NETWORK
TITLE = CALL SFC PH_EMC2_CHARGE if CHARGE running
//------------------------------------------------------------------------//
// SFC CALL   SFC CALL   SFC CALL   SFC CALL   SFC CALL   SFC CALL   SFC  //
//                                                                        //
// Call the SFC function if this is the running substate. This has to be  //
// called even if the block is not running so the SFC can process all     //
// commmands:                                                             //
//------------------------------------------------------------------------//
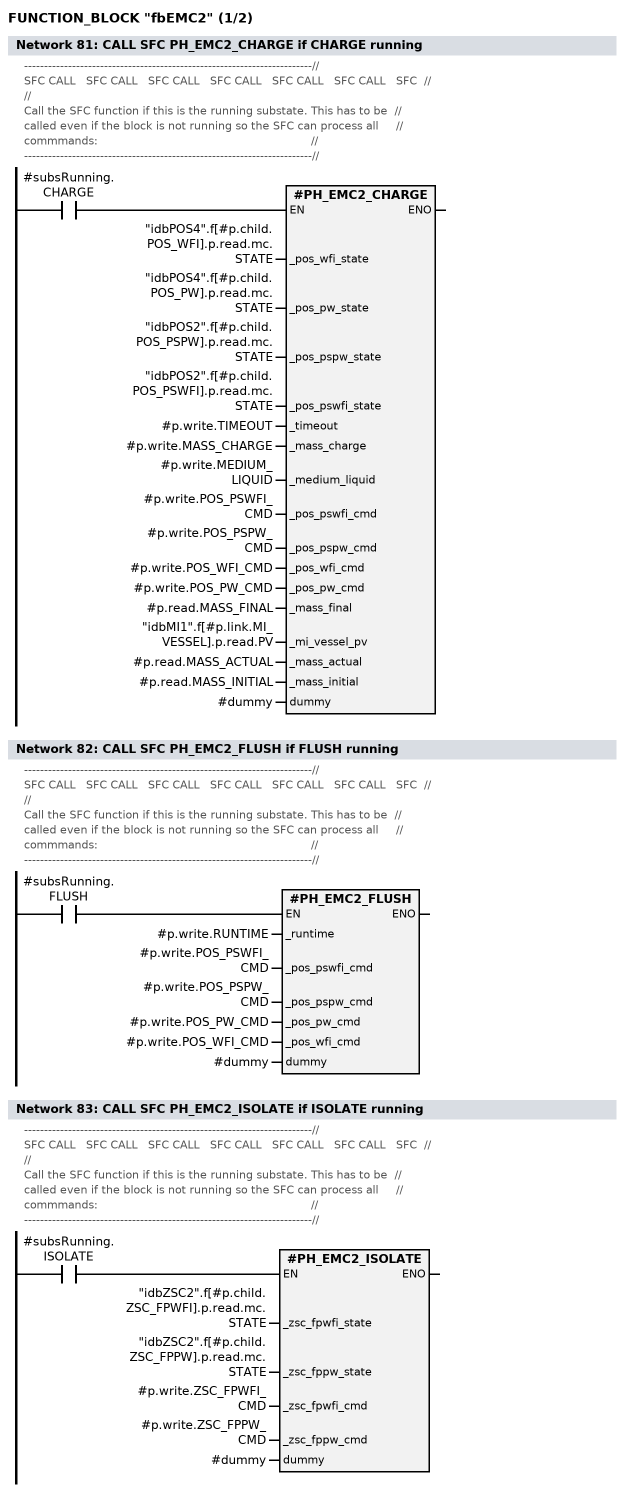
      A #subsRunning.CHARGE;
      JCN _notSFC_1_CHARGE;
      CALL #PH_EMC2_CHARGE
      (  _pos_wfi_state              := "idbPOS4".f[#p.child.POS_WFI].p.read.mc.STATE ,
         _pos_pw_state               := "idbPOS4".f[#p.child.POS_PW].p.read.mc.STATE ,
         _pos_pspw_state             := "idbPOS2".f[#p.child.POS_PSPW].p.read.mc.STATE ,
         _pos_pswfi_state            := "idbPOS2".f[#p.child.POS_PSWFI].p.read.mc.STATE ,
         _timeout                    := #p.write.TIMEOUT ,
         _mass_charge                := #p.write.MASS_CHARGE ,
         _medium_liquid              := #p.write.MEDIUM_LIQUID ,
         _pos_pswfi_cmd              := #p.write.POS_PSWFI_CMD ,
         _pos_pspw_cmd               := #p.write.POS_PSPW_CMD ,
         _pos_wfi_cmd                := #p.write.POS_WFI_CMD ,
         _pos_pw_cmd                 := #p.write.POS_PW_CMD ,
         _mass_final                 := #p.read.MASS_FINAL ,
         _mi_vessel_pv               := "idbMI1".f[#p.link.MI_VESSEL].p.read.PV ,
         _mass_actual                := #p.read.MASS_ACTUAL ,
         _mass_initial               := #p.read.MASS_INITIAL ,
         dummy                       := #dummy
      );
_notSFC_1_CHARGE:      NOP 0;
NETWORK
TITLE = CALL SFC PH_EMC2_FLUSH if FLUSH running
//------------------------------------------------------------------------//
// SFC CALL   SFC CALL   SFC CALL   SFC CALL   SFC CALL   SFC CALL   SFC  //
//                                                                        //
// Call the SFC function if this is the running substate. This has to be  //
// called even if the block is not running so the SFC can process all     //
// commmands:                                                             //
//------------------------------------------------------------------------//
      A #subsRunning.FLUSH;
      JCN _notSFC_1_FLUSH;
      CALL #PH_EMC2_FLUSH
      (  _runtime                    := #p.write.RUNTIME ,
         _pos_pswfi_cmd              := #p.write.POS_PSWFI_CMD ,
         _pos_pspw_cmd               := #p.write.POS_PSPW_CMD ,
         _pos_pw_cmd                 := #p.write.POS_PW_CMD ,
         _pos_wfi_cmd                := #p.write.POS_WFI_CMD ,
         dummy                       := #dummy
      );
_notSFC_1_FLUSH:      NOP 0;
NETWORK
TITLE = CALL SFC PH_EMC2_ISOLATE if ISOLATE running
//------------------------------------------------------------------------//
// SFC CALL   SFC CALL   SFC CALL   SFC CALL   SFC CALL   SFC CALL   SFC  //
//                                                                        //
// Call the SFC function if this is the running substate. This has to be  //
// called even if the block is not running so the SFC can process all     //
// commmands:                                                             //
//------------------------------------------------------------------------//
      A #subsRunning.ISOLATE;
      JCN _notSFC_1_ISOLATE;
      CALL #PH_EMC2_ISOLATE
      (  _zsc_fpwfi_state            := "idbZSC2".f[#p.child.ZSC_FPWFI].p.read.mc.STATE ,
         _zsc_fppw_state             := "idbZSC2".f[#p.child.ZSC_FPPW].p.read.mc.STATE ,
         _zsc_fpwfi_cmd              := #p.write.ZSC_FPWFI_CMD ,
         _zsc_fppw_cmd               := #p.write.ZSC_FPPW_CMD ,
         dummy                       := #dummy
      );
_notSFC_1_ISOLATE:      NOP 0;
NETWORK
TITLE = CALL SFC PH_EMC2_SETUP if SETUP running
//------------------------------------------------------------------------//
// SFC CALL   SFC CALL   SFC CALL   SFC CALL   SFC CALL   SFC CALL   SFC  //
//                                                                        //
// Call the SFC function if this is the running substate. This has to be  //
// called even if the block is not running so the SFC can process all     //
// commmands:                                                             //
//------------------------------------------------------------------------//
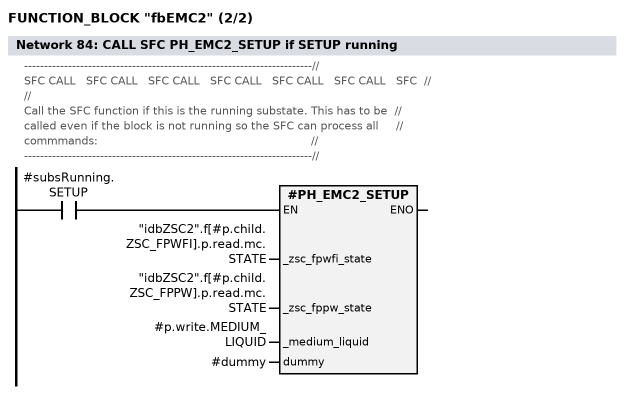
      A #subsRunning.SETUP;
      JCN _notSFC_1_SETUP;
      CALL #PH_EMC2_SETUP
      (  _zsc_fpwfi_state            := "idbZSC2".f[#p.child.ZSC_FPWFI].p.read.mc.STATE ,
         _zsc_fppw_state             := "idbZSC2".f[#p.child.ZSC_FPPW].p.read.mc.STATE ,
         _medium_liquid              := #p.write.MEDIUM_LIQUID ,
         dummy                       := #dummy
      );
_notSFC_1_SETUP:      NOP 0;

NETWORK
TITLE = Check if any Child state does not match the command
//------------------------------------------------------------------------//
// CHILD FLOWPATH STATE MISMATCH   CHILD FLOWPATH STATE MISMATCH   CHILD  //
//                                                                        //
// Check if any child flowpath device state does not match the command    //
// from this parent block if the child state grace period timer has       //
// expired. Stop checking if the first child state mismatch found:        //
//------------------------------------------------------------------------//
      A(;
      O(;
      A "alwaysHigh";
      A "idbPOS2".f[#p.child.POS_PSPW].p.write.mc.ARMED;
      A "idbPOS2".f[#p.child.POS_PSPW].p.read.mc.FLOWPATH;
      A(;
      L "idbPOS2".f[#p.child.POS_PSPW].p.read.mc.STATE;
      L #childReqCMD.POS_PSPW;
      <>I;
      );
      );
      O(;
      A "alwaysHigh";
      A "idbPOS2".f[#p.child.POS_PSWFI].p.write.mc.ARMED;
      A "idbPOS2".f[#p.child.POS_PSWFI].p.read.mc.FLOWPATH;
      A(;
      L "idbPOS2".f[#p.child.POS_PSWFI].p.read.mc.STATE;
      L #childReqCMD.POS_PSWFI;
      <>I;
      );
      );
      O(;
      A "alwaysHigh";
      A "idbPOS4".f[#p.child.POS_PW].p.write.mc.ARMED;
      A "idbPOS4".f[#p.child.POS_PW].p.read.mc.FLOWPATH;
      A(;
      L "idbPOS4".f[#p.child.POS_PW].p.read.mc.STATE;
      L #childReqCMD.POS_PW;
      <>I;
      );
      );
      O(;
      A "alwaysHigh";
      A "idbPOS4".f[#p.child.POS_WFI].p.write.mc.ARMED;
      A "idbPOS4".f[#p.child.POS_WFI].p.read.mc.FLOWPATH;
      A(;
      L "idbPOS4".f[#p.child.POS_WFI].p.read.mc.STATE;
      L #childReqCMD.POS_WFI;
      <>I;
      );
      );
      O(;
      A "alwaysHigh";
      A "idbZSC2".f[#p.child.ZSC_FPINLET].p.write.mc.ARMED;
      A "idbZSC2".f[#p.child.ZSC_FPINLET].p.read.mc.FLOWPATH;
      A(;
      L "idbZSC2".f[#p.child.ZSC_FPINLET].p.read.mc.STATE;
      L #childReqCMD.ZSC_FPINLET;
      <>I;
      );
      );
      O(;
      A "alwaysHigh";
      A "idbZSC2".f[#p.child.ZSC_FPPW].p.write.mc.ARMED;
      A "idbZSC2".f[#p.child.ZSC_FPPW].p.read.mc.FLOWPATH;
      A(;
      L "idbZSC2".f[#p.child.ZSC_FPPW].p.read.mc.STATE;
      L #childReqCMD.ZSC_FPPW;
      <>I;
      );
      );
      O(;
      A "alwaysHigh";
      A "idbZSC2".f[#p.child.ZSC_FPWFI].p.write.mc.ARMED;
      A "idbZSC2".f[#p.child.ZSC_FPWFI].p.read.mc.FLOWPATH;
      A(;
      L "idbZSC2".f[#p.child.ZSC_FPWFI].p.read.mc.STATE;
      L #childReqCMD.ZSC_FPWFI;
      <>I;
      );
      );
      );
      JCN _noMismatch;

      S #flags.childMismatch;
      JC _noResetMismatch;

_noMismatch:      NOP 0;
      R #flags.childMismatch;
      R #p.read.mc.INTIL;

_noResetMismatch:      NOP 0;

NETWORK
TITLE = If child command changed, start timer to wait for child state
//------------------------------------------------------------------------//
// CHILD STATE TIMER   CHILD STATE TIMER   CHILD STATE TIMER   CHILD STAT //
//                                                                        //
// If any child command changed then start a timer to provide a grace     //
// period to allow the child device state to match the command (e.g. to   //
// allow a valve to move from closed to opened position).                 //
// Start the child state check timer if a command changed:                //
//------------------------------------------------------------------------//
      CALL #timeCheckChildState
      {time_type := 'Time'}
      (  IN                          := #flags.childMismatch ,
         PT                          := #p.read.bmc.transTime ,
         Q                           := #timeCheckChildStateExpired ,
         ET                          := #timeCheckChildStateElapsed
      );
      NOP 0;

NETWORK
TITLE = Block errors
//------------------------------------------------------------------------//
// Set the block start perimt error status if active:                     //
//------------------------------------------------------------------------//
      AN #p.read.bmc.permitStart;
      = #p.read.err.permitStart;

  //------------------------------------------------------------------------//
  // Set the child error status if active:                                  //
  //------------------------------------------------------------------------//
      A #flags.childInterlock;
      = #p.read.err.childInterlock;

  //------------------------------------------------------------------------//
  // Set the child unavailable error status if active:                      //
  //------------------------------------------------------------------------//
      A #flags.childUnavailable;
      = #p.read.err.childUnavailable;

  //------------------------------------------------------------------------//
  // Set the child state mismatch error status if active:                   //
  //------------------------------------------------------------------------//
      A #timeCheckChildStateExpired;
      = #p.read.err.childMismatch;
      JCN _noInternalIL;
      S #p.read.mc.INTIL;
_noInternalIL:      NOP 0;

  //------------------------------------------------------------------------//
  // Set the block error flag if anything gone wrong:                       //
  //------------------------------------------------------------------------//
      O #p.read.err.childInterlock;
      O #p.read.err.childMismatch;
      O #p.read.err.childSafeState;
      O #p.read.err.childUnavailable;
      O #p.read.err.permitStart;
      = #p.read.mc.ERROR;

NETWORK
TITLE = Pack the general block alarm bits
//------------------------------------------------------------------------//
// Pack the alarm bits into an integer for the HMI to read:               //
// Alarms are arranged in the following Little Endian order...            //
// Word   1                                0                              //
// Bit    0   1   2   3   4   5   6   7    8   9  10  11  12  13  14  15  //
// Order  9  10  11  12  13  14  15  16    1   2   3   4   5   6   7   8  //
//------------------------------------------------------------------------//
//    A #p.read.err.childInterlock;
//    = #b[8];
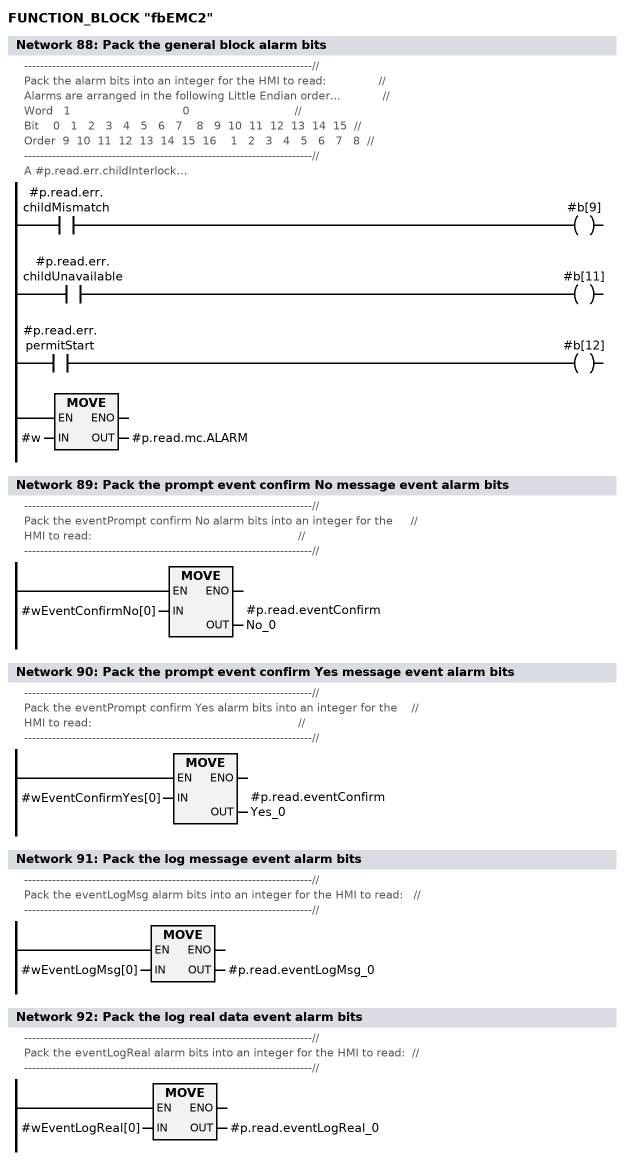
      A #p.read.err.childMismatch;
      = #b[9];
//    A #p.read.err.childSafeState;
//    = #b[10];
      A #p.read.err.childUnavailable;
      = #b[11];
      A #p.read.err.permitStart;
      = #b[12];
      L #w;
      T #p.read.mc.ALARM;

NETWORK
TITLE = Pack the prompt event confirm No message event alarm bits
//------------------------------------------------------------------------//
// Pack the eventPrompt confirm No alarm bits into an integer for the     //
// HMI to read:                                                           //
//------------------------------------------------------------------------//
      L #wEventConfirmNo[0];
      T #p.read.eventConfirmNo_0;

NETWORK
TITLE = Pack the prompt event confirm Yes message event alarm bits
//------------------------------------------------------------------------//
// Pack the eventPrompt confirm Yes alarm bits into an integer for the    //
// HMI to read:                                                           //
//------------------------------------------------------------------------//
      L #wEventConfirmYes[0];
      T #p.read.eventConfirmYes_0;

NETWORK
TITLE = Pack the log message event alarm bits
//------------------------------------------------------------------------//
// Pack the eventLogMsg alarm bits into an integer for the HMI to read:   //
//------------------------------------------------------------------------//
      L #wEventLogMsg[0];
      T #p.read.eventLogMsg_0;

NETWORK
TITLE = Pack the log real data event alarm bits
//------------------------------------------------------------------------//
// Pack the eventLogReal alarm bits into an integer for the HMI to read:  //
//------------------------------------------------------------------------//
      L #wEventLogReal[0];
      T #p.read.eventLogReal_0;


END_FUNCTION_BLOCK

